// TIA Portal V18 export
VAR_GLOBAL   // PLC tag table "Standard-Variablentabelle"
END_VAR
